INTERFACE ITF_Component_TE2_HMI EXTENDS ITF_BaseComponent_HMI

METHOD LinkComponentData : BOOL
VAR_INPUT
	stData				: REFERENCE TO ST_Component_TE2_HMI_Link;
END_VAR
END_METHOD

END_INTERFACE

(* stored: Version 1.1.0.1, ProductVersion 3.1.4024.15
   Itf ITF_Component_TE2_HMI: Id {79414b42-6e30-452f-a171-57f49a3177ac}
   Method LinkComponentData: Id {d600d72f-3bb8-4c9e-b13d-44c8805d5b73} *)
